// TIA Portal V19 export
TYPE "CTRL_MTRDIR"
   STRUCT
      status : Bool;
      sim : "UDT_SIM_MTR";
   END_STRUCT;
END_TYPE
